TYPE StepperENCStatus :
STRUCT
	LatchCValid : BOOL;
	LatchExternalValid : BOOL;
	SetCounterDone : BOOL;
	CounterUnderflow : BOOL;
	CounterOverflow : BOOL;
	ExtrapolationStall : BOOL;
	StatusInputA : BOOL;
	StatusInputB : BOOL;
	StatusInputC : BOOL;
	StatusExternLatch : BOOL;
	SyncError : BOOL;
	TxPDOToggle : BOOL;
	CounterValue : UDINT;
	LatchValue : UDINT;
END_STRUCT
END_TYPE

(* stored: Version 1.1.0.1, ProductVersion 3.1.4024.9
   DUT StepperENCStatus: Id {6d621f19-fffe-46ad-a857-c4dcd71eccf6} *)
